FUNCTION_BLOCK PUBLIC FB_Engine
VAR
	maxVelocityInternal		:	LREAL := 50.0;
	velocityInternal		:	LREAL;	
	temperatureInternal		:	INT;
END_VAR

{attribute 'monitoring' := 'variable'}
PROPERTY PUBLIC MaxVelocity : LREAL
GET
MaxVelocity := maxVelocityInternal;
END_GET
SET
maxVelocityInternal := MaxVelocity;
END_SET
END_PROPERTY

METHOD PUBLIC Start
VAR_INPUT
	nGear		:	INT := 2;
	fVelocity	:	LREAL := 8.0;
END_VAR
IF (fVelocity < MaxVelocity) THEN
	velocityInternal := fVelocity;
ELSE
	velocityInternal := MaxVelocity;
END_IF
END_METHOD

METHOD PUBLIC Stop
VAR_INPUT
END_VAR
velocityInternal := 0;
END_METHOD

{attribute 'monitoring' := 'variable'}
PROPERTY PUBLIC Temperature : INT
GET
Temperature := temperatureInternal;
END_GET
END_PROPERTY

{attribute 'monitoring' := 'variable'}
PROPERTY PUBLIC Velocity : LREAL
GET
Velocity := velocityInternal;
END_GET
END_PROPERTY

END_FUNCTION_BLOCK

(* stored: Version 1.1.0.1, ProductVersion 3.1.4020.12
   POU FB_Engine: Id {ee886422-c9f9-465c-9669-80f0cd7f24c5}, SpecialFunc None
   Property MaxVelocity: Id {5832ae5d-f51d-4b6c-87eb-563a1939fbb9}
   Get Get: Id {8f75e2ed-6d47-474d-988e-69529e92b9c9}
   Set Set: Id {abb1ec62-326c-4d9b-ba92-261e81a5ec78}
   Method Start: Id {7719b75f-dddc-4422-85ad-2e331cc1ade1}
   Method Stop: Id {bce89059-4627-457c-9768-faf38c91a607}
   Property Temperature: Id {3873a212-d323-481e-aed4-cdebb77b7820}
   Get Get: Id {12432250-c84f-4114-8c13-ade6b73ea879}
   Property Velocity: Id {346c8242-4523-47c1-8419-be4413853455}
   Get Get: Id {7ed5d34e-d8dc-4506-9902-bd51cd2c86fb} *)
